SYSTEM Test Big Computation 1
  (* Version 1.0, 2005-12-23, Goran Cengic, Chalmers *)
  DEVICE Test Device : DeviceType_not_used
    RESOURCE Test Resource : ResourceType_not_used
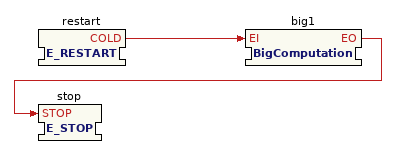
      FBS
        restart : E_RESTART;
        stop : E_STOP;
        big1 : BigComputation;
      END_FBS
      EVENT_CONNECTIONS
        restart.COLD TO big1.EI;
        big1.EO TO stop.STOP;
      END_CONNECTIONS
    END_RESOURCE
  END_DEVICE
END_SYSTEM
